FUNCTION_BLOCK TurnTableManualIProv (* Turn Table Manual Interface Provider *)
  (* Standard: 61499-2 *)
  (* Version 0.2, 2003-12-05, JHC, Rockwell Automation, Renamed from NEWCOMPFB. *)
  (* Version 0.1, 2002-01-08, JHC, Rockwell Automation, Added DLY FB as example. *)
  (* Version 0.0, 2000-05-27, JHC, Rockwell Automation *)
  (* Compiler header: package fb.rt.dasdA1.A2.TurnTable; *)
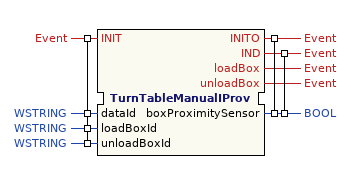
  EVENT_INPUT
    INIT WITH dataId, loadBoxId, unloadBoxId; (* Initialization Request *)
  END_EVENT
  EVENT_OUTPUT
    INITO WITH boxProximitySensor; (* Initialization Confirm *)
    IND WITH boxProximitySensor;
    loadBox;
    unloadBox;
  END_EVENT
  VAR_INPUT
    dataId : WSTRING;
    loadBoxId : WSTRING;
    unloadBoxId : WSTRING;
  END_VAR
  VAR_OUTPUT
    boxProximitySensor : BOOL;
  END_VAR
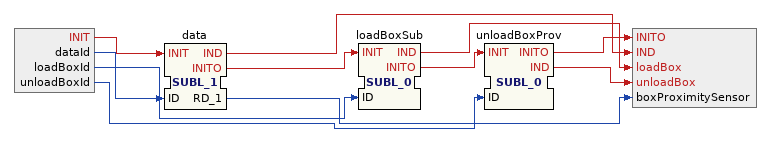
  FBS
    loadBoxSub : SUBL_0;
    data : SUBL_1;
    unloadBoxProv : SUBL_0;
  END_FBS
  EVENT_CONNECTIONS
    loadBoxSub.IND TO loadBox;
    INIT TO data.INIT;
    data.IND TO IND;
    data.INITO TO loadBoxSub.INIT;
    loadBoxSub.INITO TO unloadBoxProv.INIT;
    unloadBoxProv.INITO TO INITO;
    unloadBoxProv.IND TO unloadBox;
  END_CONNECTIONS
  DATA_CONNECTIONS
    loadBoxId TO loadBoxSub.ID;
    dataId TO data.ID;
    data.RD_1 TO boxProximitySensor;
    unloadBoxId TO unloadBoxProv.ID;
  END_CONNECTIONS
END_FUNCTION_BLOCK
